// TIA Portal project "NutNhan" (V14)

(* hardware
DEVICE "S7-1200 station_1"  S7-1200 Station
   slot 0: "Rack_0"  S7-1200 Rack  Rack  V1.0
   slot 1: "PLC_1"  CPU 1214C DC/DC/Rly  6ES7 214-1HG40-0XB0  V4.2
*)

// ===== PLC "PLC_1"  CPU 1214C DC/DC/Rly =====

VAR_GLOBAL   // PLC tag table "Default tag table"
   "Tag_1" AT %M0.0 : Bool;
   "Tag_2" AT %Q0.0 : Bool;
   "Tag_3" AT %Q0.1 : Bool;
   "Tag_4" AT %Q0.2 : Bool;
   "Tag_5" AT %M0.1 : Bool;
   "Tag_6" AT %M0.2 : Bool;
   "Tag_7" AT %M0.3 : Bool;
END_VAR

ORGANIZATION_BLOCK "Main"   // OB1, LAD, ProgramCycle
TITLE = "Main Program Sweep (Cycle)"
{ S7_Optimized_Access := 'TRUE' }
VERSION : 0.1
   VAR_INPUT
      Initial_Call : Bool;   // Initial call of this OB
      Remanence : Bool;   // =True, if remanent data are available
   END_VAR
BEGIN

REGION Network 1
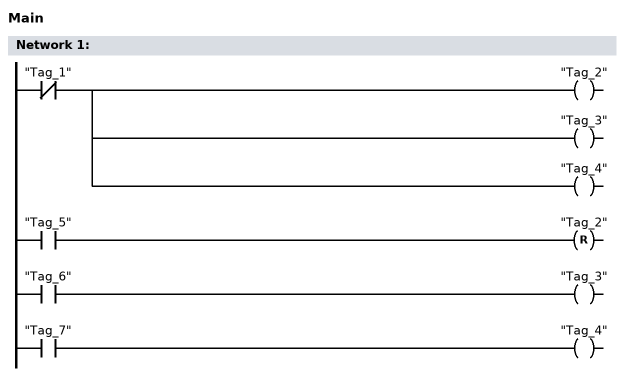
   RUNG wire#powerrail
      I_Contact( "Tag_1" )
      wire#w1
      Coil( "Tag_2" )
   END_RUNG
   RUNG wire#w1
      Coil( "Tag_3" )
   END_RUNG
   RUNG wire#w1
      Coil( "Tag_4" )
   END_RUNG
   RUNG wire#powerrail
      Contact( "Tag_5" )
      R_Coil( "Tag_2" )
   END_RUNG
   RUNG wire#powerrail
      Contact( "Tag_6" )
      Coil( "Tag_3" )
   END_RUNG
   RUNG wire#powerrail
      Contact( "Tag_7" )
      Coil( "Tag_4" )
   END_RUNG
   // the same network as SCL:
   "Tag_2" := NOT "Tag_1";
   "Tag_3" := NOT "Tag_1";
   "Tag_4" := NOT "Tag_1";
   IF "Tag_5" THEN "Tag_2" := FALSE; END_IF;
   "Tag_3" := "Tag_6";
   "Tag_4" := "Tag_7";
END_REGION
END_ORGANIZATION_BLOCK